// TIA Portal project "project_counter_application" (V16)

(* hardware
DEVICE "S7-1200 station_1"  S7-1200 Station
   slot 0: "Rack_0"  S7-1200 Rack  Rack  V1.0
   slot 1: "PLC_1"  CPU 1214C DC/DC/Rly  6ES7 214-1HG40-0XB0  V4.4
*)

// ===== PLC "PLC_1"  CPU 1214C DC/DC/Rly =====

VAR_GLOBAL   // PLC tag table "Default tag table"
   "START BUT" AT %I0.0 : Bool;
   "MOTOR-2" AT %Q0.1 : Bool;
   "MOTOR-3" AT %Q0.2 : Bool;
   "MOTOR-1" AT %Q0.0 : Bool;
   "RESETLE" AT %M30.0 : Bool;
   "TERMİK 1" AT %I0.2 : Bool;
   "TERMİK 2" AT %I0.3 : Bool;
   "TERMİK 3" AT %I0.4 : Bool;
END_VAR

// folder: System blocks/Program resources

DATA_BLOCK "COUNTER 1"   // DB1
{ S7_Optimized_Access := 'TRUE' }
AUTHOR : Simatic
FAMILY : IEC
NAME : CNTR
VERSION : 1.0
// stored: InstanceOfName IEC_COUNTER
"IEC_COUNTER"
BEGIN
END_DATA_BLOCK

DATA_BLOCK "COUNTER 2"   // DB2
{ S7_Optimized_Access := 'TRUE' }
AUTHOR : Simatic
FAMILY : IEC
NAME : CNTR
VERSION : 1.0
// stored: InstanceOfName IEC_COUNTER
"IEC_COUNTER"
BEGIN
END_DATA_BLOCK

DATA_BLOCK "COUNTER 3"   // DB3
{ S7_Optimized_Access := 'TRUE' }
AUTHOR : Simatic
FAMILY : IEC
NAME : CNTR
VERSION : 1.0
// stored: InstanceOfName IEC_COUNTER
"IEC_COUNTER"
BEGIN
END_DATA_BLOCK

DATA_BLOCK "COUNTER 4"   // DB4
{ S7_Optimized_Access := 'TRUE' }
AUTHOR : Simatic
FAMILY : IEC
NAME : CNTR
VERSION : 1.0
// stored: InstanceOfName IEC_COUNTER
"IEC_COUNTER"
BEGIN
END_DATA_BLOCK

// folder: (top level)

ORGANIZATION_BLOCK "Main"   // OB1, LAD, ProgramCycle
TITLE = "Main Program Sweep (Cycle)"
{ S7_Optimized_Access := 'TRUE' }
VERSION : 0.1
   VAR_INPUT
      Initial_Call : Bool;   // Initial call of this OB
      Remanence : Bool;   // =True, if remanent data are available
   END_VAR
BEGIN

REGION Network 1
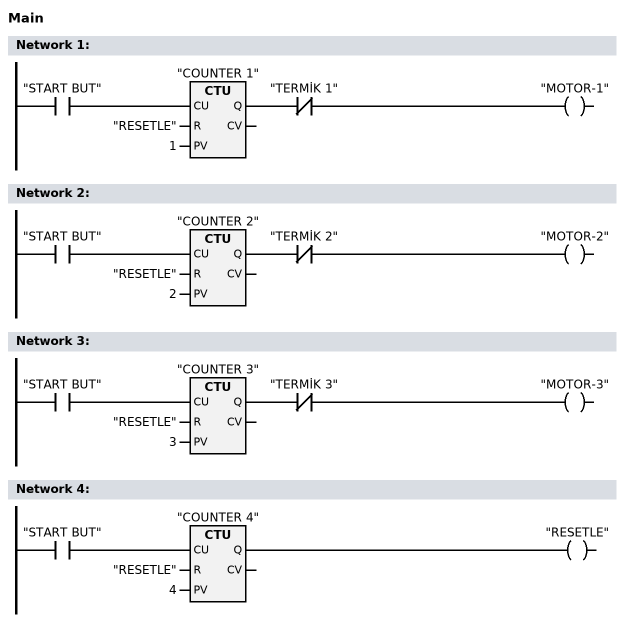
   "COUNTER 1".CTU(CU := "START BUT", R := "RESETLE", PV := 1);
   "MOTOR-1" := "COUNTER 1".Q AND NOT "TERMİK 1";
END_REGION

REGION Network 2
   "COUNTER 2".CTU(CU := "START BUT", R := "RESETLE", PV := 2);
   "MOTOR-2" := "COUNTER 2".Q AND NOT "TERMİK 2";
END_REGION

REGION Network 3
   "COUNTER 3".CTU(CU := "START BUT", R := "RESETLE", PV := 3);
   "MOTOR-3" := "COUNTER 3".Q AND NOT "TERMİK 3";
END_REGION

REGION Network 4
   "COUNTER 4".CTU(CU := "START BUT", R := "RESETLE", PV := 4);
   "RESETLE" := "COUNTER 4".Q;
END_REGION
END_ORGANIZATION_BLOCK